FUNCTION_BLOCK FB_PTOStepperMoveRel
VAR_INPUT
	bExecute	: BOOL;
	bStop		: BOOL;
	nSteps		: INT;
	nSpeed		: UINT;	//Steps/sec	
END_VAR
VAR_OUTPUT
	bBusy		: BOOL;
END_VAR
VAR_IN_OUT
	pPTOStepperRef : POINTER TO ST_PTOStepperRef;	
END_VAR
VAR
	nState : USINT;
	nSpeedIntern: INT;
END_VAR

IF bExecute THEN
	CASE nState OF
		0:	//Prepare
			IF bStop THEN
				RETURN;
			END_IF
			
			bBusy := TRUE;
			IF nSteps < 0 THEN
				//CCW Drehung -> muss Richtung "0" drehen -> auf Counter "0" oder Counter underflow abfragen
				pPTOStepperRef^.nSetCounterValue := INT_TO_UINT(ABS(nSteps));
				nSpeedIntern := -UINT_TO_INT(nSpeed);
			ELSIF nSteps > 0 THEN
				//CW Drehung -> muss Richtung "0" drehen -> auf Counter >= SetCounter oder Counter overflow abfragen
				pPTOStepperRef^.nSetCounterValue := 0;
				nSpeedIntern := UINT_TO_INT(nSpeed);
			ELSE
				bBusy := FALSE;
				nState := 80;
				RETURN;
			END_IF
			pPTOStepperRef^.bSetCounter := TRUE;
			nState := 1;
			
		1:	//Start
			IF bStop THEN
				bBusy := FALSE;
				nState := 80;
				RETURN;
			END_IF
			IF pPTOStepperRef^.nSetCounterValue = pPTOStepperRef^.nCountervalue THEN
				pPTOStepperRef^.bSetCounter := FALSE;
				MEMCPY(ADR(pPTOStepperRef^.nFrequencyValue),ADR(nSpeedIntern),2);
				nState := 2;
			END_IF
			
		2:	//Waiting for target reached
			IF bStop OR
					 	//CCW Drehung -> abwärts zählen -> auf Counter "0" oder Counter underflow abfragen
						((nSteps < 0) AND ((pPTOStepperRef^.nCountervalue = 0) OR pPTOStepperRef^.bCounterUnderflow))
					 OR
					 	//CW Drehung -> aufwärts zählen -> auf Counter >= SetCounter oder Counter overflow abfragen
						((nSteps > 0) AND ((pPTOStepperRef^.nCountervalue >= INT_TO_UINT(ABS(nSteps))) OR pPTOStepperRef^.bCounterUnderflow))THEN
						
				pPTOStepperRef^.nFrequencyValue := 0;
				nState := 3;
			END_IF
			
		3:	//Wartezyklus
			bBusy := FALSE;
	END_CASE
ELSE
	nState := 0;
	bBusy := FALSE;
END_IF

END_FUNCTION_BLOCK

(* stored: Version 1.1.0.1, ProductVersion 3.1.4020.12
   POU FB_PTOStepperMoveRel: Id {fbe886f9-1aa1-4fa2-b768-f66bd8b5bd7d}, SpecialFunc None *)
